FUNCTION_BLOCK ResolveTestCompFbt
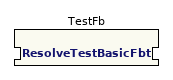
  FBS
    TestFb : ResolveTestBasicFbt;
  END_FBS
END_FUNCTION_BLOCK
